(* PLC project Unnamed, Unknown Unnamed 1 *)
(* stored: creationDateTime 2025-11-05T10:34:14, modificationDateTime 2025-11-05T10:53:17 *)

PROGRAM main
  VAR
    Mission1 : BOOL := False;
    Mission2 : BOOL := False;
    Mission1_Done : BOOL := False;
    Mission1_Start : BOOL := False;
    Mission2_Done : BOOL := False;
    Mission2_Start : BOOL := False;
    AutoRunning : BOOL := False;
    NoMission : BOOL := False;
  END_VAR

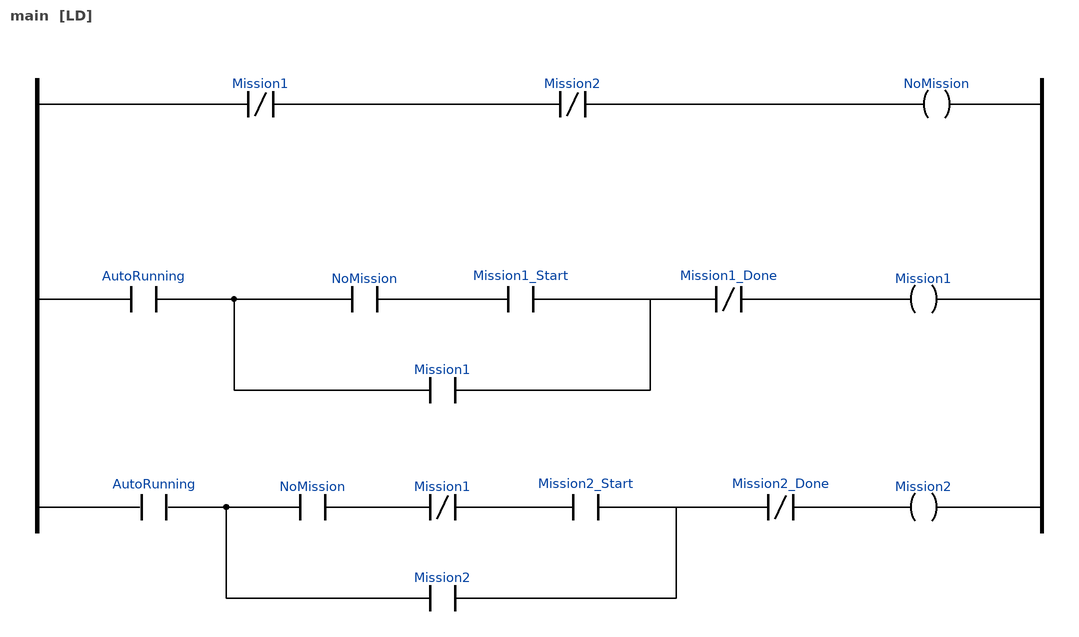
(* LD diagram, written out as Structured Text *)
NoMission := NOT Mission1 AND NOT Mission2;
Mission1 := AutoRunning AND (NoMission AND Mission1_Start OR Mission1) AND NOT Mission1_Done;
Mission2 := AutoRunning AND (NoMission AND NOT Mission1 AND Mission2_Start OR Mission2) AND NOT Mission2_Done;
END_PROGRAM

CONFIGURATION Config0
  RESOURCE Res0 ON PLC
    TASK task0(INTERVAL := T#20ms, PRIORITY := 0);
    PROGRAM instance0 WITH task0 : main;
  END_RESOURCE
END_CONFIGURATION
